// TwinCAT 3 PLC project Nepionic_Motion_Test
// ProgramVersion: 3.1.4026.19
// libraries:
//   Nepionic_Core, * (Nepionic)
//   [Nepionic_Motion], * (Nepionic)
//   Tc2_System, * (Beckhoff Automation GmbH)
//   Tc3_Module, * (Beckhoff Automation GmbH)
// project tree:
//   Programs/ Test.TcPOU
//   Tasks/ TestTask.TcTTO
// real-time tasks:
//   TASK TestTask: cycle T#10ms, priority 20, ADS port 350
// motion (NC):
//   TASK NC-Task 1 SAF: cycle T#2ms, priority 4, ADS port 501
//   TASK NC-Task 1 SVB: cycle T#10ms, priority 8, ADS port 511
//   AXIS Axis 1 (id 1)
//     OtherSettings: AllowMotionCmdToSlave=true
//     encoder EncType=1
//     drive DrvType=5
//       Analog: TorqueSetpointScale=10, ScaleFactorActTorque=0.1
//       TimeComp: TaskDelayCycles=1
//     controller CtrType=1
//       CtrPara: PriorControlFactor=1
//         Observer: BandWidth=20
//   AXIS Axis 2 (id 2)
//     OtherSettings: AllowMotionCmdToSlave=true
//     encoder EncType=1
//     drive DrvType=5
//       Analog: TorqueSetpointScale=10, ScaleFactorActTorque=0.1
//     controller CtrType=1
//       CtrPara: PriorControlFactor=1
//         Observer: BandWidth=20
// variable links:
//   Nepionic_Motion_Test Instance <-> NC-Task 1 SAF/Axes/Axis 1
//     TestTask Inputs/Test.axis1.axis_ref.NcToPlc <-> Outputs/ToPlc
//     TestTask Outputs/Test.axis1.axis_ref.PlcToNc <-> Inputs/FromPlc
//   Nepionic_Motion_Test Instance <-> NC-Task 1 SAF/Axes/Axis 2
//     TestTask Inputs/Test.axis2.axis_ref.NcToPlc <-> Outputs/ToPlc
//     TestTask Outputs/Test.axis2.axis_ref.PlcToNc <-> Inputs/FromPlc

CONFIGURATION Nepionic_Motion_Test
    RESOURCE PLC ON TwinCAT3
        TASK TestTask(INTERVAL := T#10ms, PRIORITY := 20);
        PROGRAM Test WITH TestTask : Test;
    END_RESOURCE
END_CONFIGURATION

// ---- Programs/Test.TcPOU
PROGRAM Test
VAR
	axis1 : Mc2Axis;
	axis2 : Mc2Axis;
	
	busy : BOOL;
	active : BOOL;
	done : BOOL;
	aborted : BOOL;
	error : BOOL;
	error_id : UDINT;
	
	enable: BOOL;
	disable: BOOL;
	reset: BOOL;
	halt: BOOL;
	stop: BOOL;

	jog_forward : BOOL;
	jog_backwards : BOOL;
	
	start_move1 : BOOL;
	start_move2 : BOOL;
	
	start_homing : BOOL;
	
	gear_in : BOOL;
	gear_in_numerator : LREAL := 1;
	gear_in_denominator : UINT := 1;
	
	gear_out : BOOL;
	
	move1_command : MotionCommand;
	move2_command : MotionCommand;
	halt_command : MotionCommand;
	stop_command : MotionCommand;
	gear_in_command : AsyncCommand;
	gear_out_command : AsyncCommand;
	
	move_builder : DefaultMotionBuilder;
END_VAR

axis1.CyclicCall();
axis2.CyclicCall();

error := axis1.IsErrored;
error_id := axis1.ErrorId;

IF enable THEN
	enable := FALSE;
	//axis1.Enable(AxisBufferMode.Buffered);
	axis1.Enable();
	axis1.EnablePositive();
	axis1.EnableNegative();
	axis2.Enable();
	axis2.EnablePositive();
	axis2.EnableNegative();
END_IF

IF disable THEN
	disable := FALSE;
	axis1.Disable();
END_IF

IF reset THEN
	reset := FALSE;
	axis1.Reset();
	axis2.Reset();
END_IF

IF halt THEN
	halt := FALSE;
	IF halt_command = 0 THEN
		halt_command := move_builder
			.Reset()
			.BuildHaltCommand(axis1);
	END_IF
	halt_command.Execute();
END_IF

IF stop THEN
	stop := FALSE;
	IF stop_command = 0 THEN
		stop_command := move_builder
			.Reset()
			.BuildStopCommand(axis1);
	END_IF
	stop_command.Execute();
END_IF

IF jog_forward THEN
	//axis1.JogForward(100);
ELSIF jog_backwards THEN
	//axis1.JogBackwards(100);
ELSE
	// Don't like this, since jogging now acts like MC_MoveVelocity
	// although I guess that is what it is exactly
	//axis1.StopJogging();
END_IF

IF start_homing THEN
	start_homing := FALSE;
	(*axis1.HomingBuilder()
		.Position(homePosition)
		.BuildDirectHomingCommand()
		.Execute(homingFeedback)
		.ThenRelease();*)
	(*command := axis1.HomingBuilder()
		.Position(homePosition)
		.Cam(homeCam)
		.ReferenceMode(EncoderReferenceMode.PLCCam)
		.BuildDefaultHomingCommand();*)
END_IF

(*IF setPositionAbsolute THEN
	setPositionAbsolute := FALSE;
	axis1.SetPositionAbsolute(setPositionValue);
END_IF*)

(*IF setPositionRelative THEN
	setPositionRelative := FALSE;
	axis1.SetPositionRelative(setPositionValue);
END_IF*)

IF start_move1 THEN
	start_move1 := FALSE;
	IF move1_command = 0 THEN
		move1_command := move_builder
			.Reset()
			.Position(1000)
			.Velocity(101)
			.BufferMode(MotionBufferMode.Buffered)
			.BuildMoveAbsoluteCommand(axis1);
	END_IF
	move1_command.Execute();
END_IF

IF start_move2 THEN
	start_move2 := FALSE;
	IF move2_command = 0 THEN
		move2_command := move_builder
			.Reset()
			.Distance(1000)
			.Velocity(100)
			.BuildMoveRelativeCommand(axis1);
	END_IF
	move2_command.Execute();
END_IF

IF gear_in THEN
	gear_in := FALSE;
	IF gear_in_command = 0 THEN
		gear_in_command := move_builder
			.RatioNumerator(gear_in_numerator)
			.RatioDenominator(gear_in_denominator)
			.BuildGearInCommand(axis1, axis2);
	END_IF
	gear_in_command.Execute();
END_IF

IF gear_out THEN
	gear_out := FALSE;
	IF gear_out_command = 0 THEN
		gear_out_command := move_builder
			.BuildGearOutCommand(axis2);
	END_IF
	gear_out_command.Execute();
END_IF

IF move1_command <> 0 THEN
	move1_command.CyclicCall();

	busy := move1_command.Busy;
	active := move1_command.Active;
	done := move1_command.Done;
	aborted := move1_command.Aborted;
	error := move1_command.Error;
	error_id := move1_command.ErrorId;
END_IF

IF move2_command <> 0 THEN
	move2_command.CyclicCall();
END_IF

IF halt_command <> 0 THEN
	halt_command.CyclicCall();
END_IF

IF stop_command <> 0 THEN
	stop_command.CyclicCall();
END_IF

IF gear_in_command <> 0 THEN
	gear_in_command.CyclicCall();
END_IF

IF gear_out_command <> 0 THEN
	gear_out_command.CyclicCall();
END_IF

END_PROGRAM
